INTERFACE I_VisionMode_Base EXTENDS I_CH_Object, I_VisionMode_StatusOnly, __SYSTEM.IQueryInterface

METHOD LinkComponents : HRESULT
VAR_INPUT
	ipVisionSystem				: I_VisionSystem;
	ipCameraController 			: I_CameraController_Base;
	ipImageProvider 			: I_ImageProvider_Base;	
	ipIlluminationController1 : I_IlluminationController_Base;
	ipIlluminationController2 : I_IlluminationController_Base;
END_VAR
END_METHOD

{attribute 'monitoring' := 'call'}
// Name or description of this mode
PROPERTY Name : STRING
GET
END_GET
END_PROPERTY

END_INTERFACE

(* stored: Version 1.1.0.1, ProductVersion 3.1.4024.12
   Itf I_VisionMode_Base: Id {49c36f49-4e97-429e-94cd-b3e214e845f8}
   Method LinkComponents: Id {418f4974-c676-414c-b2a9-155325073295}
   Property Name: Id {051c6680-8ae9-4120-973c-aed51f4eec58}
   Get Get: Id {bfd0726f-80ba-493e-9092-011919a94e6f} *)
